(* IEC 61131-3 sources: ATCMcontrol_Engineering/src/TargetBase/Libs/ATCM_IEC1131_3/table_29, 9 files *)

(* ---- CONCAT.st ---- *)
FUNCTION CONCAT : ANY_STRING
VAR_INPUT
    IN1 : ANY_STRING;
END_VAR
VAR_IN_EXT
    IN2 : ANY_STRING;
END_VAR

overload STRING(STRING,STRING,...) inline { STDLIB(ConcatString) }

END_FUNCTION

(* ---- DELETE.st ---- *)
FUNCTION DELETE : ANY_STRING
VAR_INPUT
    IN : ANY_STRING;
    L : ANY_INT;
    P : ANY_INT;
END_VAR

overload STRING(STRING,         INT,         INT) inline{ STDLIB(DeleteString_int)}
overload STRING(STRING, DINT to INT, DINT to INT) inline{ STDLIB(DeleteString_int)}

END_FUNCTION

(* ---- FIND.st ---- *)
FUNCTION FIND : ANY_INT
VAR_INPUT
    IN1 : ANY_STRING;
    IN2 : ANY_STRING;
END_VAR

overload INT        (STRING, STRING) inline{ STDLIB(FindString_int) }
overload INT to DINT(STRING, STRING) inline{ STDLIB(FindString_int) }

END_FUNCTION

(* ---- INSERT.st ---- *)
FUNCTION INSERT : ANY_STRING
VAR_INPUT
    IN1 : ANY_STRING;
    IN2 : ANY_STRING;
    P : ANY_INT;
END_VAR

overload STRING(STRING, STRING,         INT) inline{ STDLIB(InsertString_int)}
overload STRING(STRING, STRING, DINT to INT) inline{ STDLIB(InsertString_int)}

END_FUNCTION

(* ---- LEFT.st ---- *)
FUNCTION LEFT : ANY_STRING
VAR_INPUT
    IN : ANY_STRING;
    L : ANY_INT;
END_VAR

overload STRING(STRING, INT)          inline{ STDLIB(LeftString_int) }
overload STRING(STRING, DINT to INT)  inline{ STDLIB(LeftString_int) }

END_FUNCTION

(* ---- LEN.st ---- *)
FUNCTION LEN : ANY_INT
VAR_INPUT
    IN : STRING;
END_VAR

overload INT        (STRING) inline { STDLIB(strlen_int) }
overload INT to DINT(STRING) inline { STDLIB(strlen_int) }

END_FUNCTION

(* ---- MID.st ---- *)
FUNCTION MID : ANY_STRING
VAR_INPUT
    IN : ANY_STRING;
    L : ANY_INT;
    P : ANY_INT;
END_VAR

overload STRING(STRING,         INT,         INT) inline{ STDLIB(MidString_int) }
overload STRING(STRING, DINT to INT, DINT to INT) inline{ STDLIB(MidString_int) }

END_FUNCTION

(* ---- REPLACE.st ---- *)
FUNCTION REPLACE : ANY_STRING
VAR_INPUT
    IN1 : ANY_STRING;
    IN2 : ANY_STRING;
    L : ANY_INT;
    P : ANY_INT;
END_VAR

overload STRING(STRING,STRING, INT,INT)                  inline{ STDLIB(ReplaceString_int) }
overload STRING(STRING,STRING, DINT to INT ,DINT to INT) inline{ STDLIB(ReplaceString_int) }

END_FUNCTION

(* ---- RIGHT.st ---- *)
FUNCTION RIGHT : ANY_STRING
VAR_INPUT
    IN : ANY_STRING;
    L : ANY_INT;
END_VAR

overload STRING(STRING,         INT) inline{ STDLIB(RightString_int) }
overload STRING(STRING, DINT to INT) inline{ STDLIB(RightString_int) }

END_FUNCTION
